TYPE ST_TestsuiteOptions :
STRUCT
		bAbortOnError:			BOOL;
END_STRUCT
END_TYPE

(* stored: Version 1.1.0.1
   DUT ST_TestsuiteOptions: Id {6fbd3cc6-28e8-07e8-0647-7149a51c793f} *)
